INTERFACE ITF_PackMLV2

{warning 'add method implementation '}
METHOD Abort : BOOL
END_METHOD

{warning 'add method implementation '}
METHOD Auto : BOOL
END_METHOD

{warning 'add method implementation '}
METHOD Clear : BOOL
END_METHOD

{warning 'add method implementation '}
METHOD Hold : BOOL
END_METHOD

{warning 'add method implementation '}
METHOD Manueel : BOOL
END_METHOD

{warning 'add method implementation '}
METHOD Reset : BOOL
END_METHOD

{warning 'add method implementation '}
METHOD Start : BOOL
END_METHOD

{warning 'add property implementation'}
PROPERTY State : E_State_PackML
GET
END_GET
END_PROPERTY

{warning 'add method implementation '}
METHOD Stop : BOOL
END_METHOD

{warning 'add method implementation '}
METHOD Suspend : BOOL
END_METHOD

{warning 'add method implementation '}
METHOD Unhold : BOOL
END_METHOD

{warning 'add method implementation '}
METHOD Unsuspend : BOOL
END_METHOD

{warning 'add method implementation '}
METHOD ZeroAllVar : BOOL
END_METHOD

END_INTERFACE

(* stored: Version 1.1.0.1, ProductVersion 3.1.4024.12
   Itf ITF_PackMLV2: Id {f36d244c-592b-4934-bf10-34d2733c2b69}
   Folder Methods: Id {ddcff743-9172-48a1-aa3f-2923a4e5a717}
   Folder Properties: Id {724ddd69-9bdd-4634-bed6-92d3b4d9f721}
   Method Abort: Id {b3cd85b6-e815-44d2-a833-35dd873cf33b}
   Method Auto: Id {8aa48e67-7f30-4c5a-b97f-486f6632b37c}
   Method Clear: Id {3a26b058-50b0-465e-b7e1-a5b6d62d326f}
   Method Hold: Id {01ce3460-6cda-44cc-91f5-e074be119b85}
   Method Manueel: Id {adbf9fec-d566-4583-978e-dd89ec08d0e3}
   Method Reset: Id {1977f694-ca78-4817-ad19-a0a555353a1e}
   Method Start: Id {a0fbca64-94bc-4799-988a-fc473354b945}
   Property State: Id {4c1cce19-aa90-4f9c-a75c-2ad4ca3a0a0f}
   Get Get: Id {df876be8-4d8b-43f1-be61-980e51c73cf5}
   Method Stop: Id {16863f13-c902-43be-8cf4-75f2a86c8c55}
   Method Suspend: Id {a9332f93-571d-4221-be3c-a212b613c2a0}
   Method Unhold: Id {0e3af376-253f-47b1-910f-f964932f88e9}
   Method Unsuspend: Id {1ab7fc9b-3f30-4613-b7ed-d67b7c48f862}
   Method ZeroAllVar: Id {fa5a6ea3-8212-4ee1-ac13-6ed8136e4ea7} *)
